// TIA Portal project "XC221_TRABALHO_FINAL" (V13)

(* hardware
DEVICE "S7-1200 station_1"  SIMATIC 1200-Station
   slot 0: "S7-1200 rack"  Rack  V1.0
   slot 1: "PLC_123"  CPU 1214C DC/DC/DC  6ES7 214-1AG31-0XB0  V3.0
   slot 3: "AQ1 x 12 bits"  6ES7 232-4HA30-0XB0  V1.0
*)

// ===== PLC "PLC_123"  CPU 1214C DC/DC/DC =====
// protected blocks, not shown: "EASYPI", "MEMRST"

VAR_GLOBAL   // PLC tag table "Default tag table"
   "System_Byte" AT %MB1 : Byte;
   "FirstScan" AT %M1.0 : Bool;   // Primeiro Scan do sistema
   "DiagStatusUpdate" AT %M1.1 : Bool;
   "AlwaysTRUE" AT %M1.2 : Bool;   // Usado para manter o sistema ligado sempre
   "AlwaysFALSE" AT %M1.3 : Bool;   // Usado para manter o sistema desligado sempre
   "Clock_Byte" AT %MB0 : Byte;
   "Clock_10Hz" AT %M0.0 : Bool;
   "Clock_5Hz" AT %M0.1 : Bool;
   "Clock_2.5Hz" AT %M0.2 : Bool;
   "Clock_2Hz" AT %M0.3 : Bool;
   "Clock_1.25Hz" AT %M0.4 : Bool;
   "Clock_1Hz" AT %M0.5 : Bool;
   "Clock_0.625Hz" AT %M0.6 : Bool;
   "Clock_0.5Hz" AT %M0.7 : Bool;
END_VAR

VAR_GLOBAL   // PLC tag table "01- Entradas Digitais"
   "DIn_GERAL_Emerge" AT %I0.0 : Bool;   // Ativa condição de emergência
   "DIn_GERAL_Rearma" AT %I0.1 : Bool;   // Rearma defeitos
   "DIn_GERAL_SelLoc" AT %I0.2 : Bool;   // Seleciona local (válvula e ventiladores)
   "DIn_VS101_Abre" AT %I0.3 : Bool;   // Botão abre válvula
   "DIn_VS101_Fecha" AT %I0.4 : Bool;   // Botão fecha válvula
   "DIn_VT101_LigDsg" AT %I0.5 : Bool;   // Botao liga/desliga ventilador 1
   "DIn_VT102_LigDsg" AT %I0.6 : Bool;   // Botao liga/desliga ventilador 2
   "DIn_BA101_DisjOff" AT %I0.7 : Bool;   // Disjuntor da bomba desarmado
END_VAR

VAR_GLOBAL   // PLC tag table "02- Saidas Digitais"
   "DOu_VS101_Abre" AT %Q0.0 : Bool;   // Abre válvula (energiza)
   "DOu_VT101_Liga" AT %Q0.1 : Bool;   // Liga ventilador 1 (energiza)
   "DOu_VT102_Liga" AT %Q0.2 : Bool;   // Liga ventilador 2 (energiza)
END_VAR

VAR_GLOBAL   // PLC tag table "03-Entradas Analogicas"
   "AIn_LT101_Nivel" AT %IW64 : UInt;   // Nível de água no tanque [bruto]
END_VAR

VAR_GLOBAL   // PLC tag table "04-Saidas Analogicas"
   "AOu_BA101_VelBmb" AT %QW64 : UInt;   // Velocidade da bomba [bruto]
END_VAR

VAR_GLOBAL   // PLC tag table "05-Comandos"
   "Cmd_GERAL_Rearma" AT %M101.0 : Bool;   // Rearma defeitos
   "Cmd_VS101_Abre" AT %M102.0 : Bool;   // Abre válvula
   "Cmd_VS101_Fecha" AT %M102.1 : Bool;   // Fecha válvula
   "Cmd_VT101_Liga" AT %M103.0 : Bool;   // Liga ventilador 1
   "Cmd_VT101_Deslig" AT %M103.1 : Bool;   // Desliga ventilador 1
   "Cmd_VT101_HorRst" AT %M103.2 : Bool;   // Zera horímetro do ventilador 1
   "Cmd_VT102_Liga" AT %M104.0 : Bool;   // Liga ventilador 2
   "Cmd_VT102_Deslig" AT %M104.1 : Bool;   // Desliga ventilador 2
   "Cmd_VT102_HorRst" AT %M104.2 : Bool;   // Zera horímetro do ventilador 2
   "Cmd_BA101_Liga" AT %M108.0 : Bool;   // Liga bomba
   "Cmd_BA101_Deslig" AT %M108.1 : Bool;   // Desliga bomba
   "Cmd_BA101_HorRst" AT %M108.2 : Bool;   // Zera horímetro da bomba
   "Cmd_BA101_SelMan" AT %M108.3 : Bool;   // Seleciona modo “Manual” da bomba
   "Cmd_BA101_SelAut" AT %M108.4 : Bool;   // Seleciona modo “Automático” da bomba
   "Cmd_BA101_SelPID" AT %M108.5 : Bool;   // Seleciona modo “PID” da bomba
   "Cmd BA101 SelOnOff" AT %M108.6 : Bool;   // Seleciona modo “On/Off” da bomba
END_VAR

VAR_GLOBAL   // PLC tag table "06-Estados"
   "Stt_GERAL_LocSel" AT %M201.0 : Bool;   // Local selecionado (válvula e ventiladores)
   "Stt_VS101_Aberta" AT %M202.0 : Bool;   // Válvula aberta (energizada)
   "Stt_VT101_Ligado" AT %M203.0 : Bool;   // Ventilador 1 ligado
   "Stt_VT101_Defeito" AT %M203.1 : Bool;   // Ventilador 1 com defeito
   "Stt_VT102_Ligado" AT %M204.0 : Bool;   // Ventilador 2 ligado
   "Stt_VT102_Defeito" AT %M204.1 : Bool;   // Ventilador 2 com defeito
   "Stt_LC101_LigBmb" AT %M206.0 : Bool;   // Solicitação do controlador On/Off para ligar bomba
   "Stt_BA101_Ligada" AT %M208.0 : Bool;   // Bomba ligada
   "Stt_BA101_Defeito" AT %M208.1 : Bool;   // Bomba com defeito
   "Stt_BA101_Bloq" AT %M208.2 : Bool;   // Bomba bloqueada
   "Stt_BA101_ManSel" AT %M208.3 : Bool;   // Bomba em modo “Manual”
   "Stt_BA101_PIDSel" AT %M208.4 : Bool;   // Bomba em modo “PID”
END_VAR

VAR_GLOBAL   // PLC tag table "07-Alarmes"
   "Alr_GERAL_Emerge" AT %M301.0 : Bool;   // Condição de emergência ativada
   "Alr_VT101_HorFim" AT %M303.0 : Bool;   // Ventilador 1 com horas esgotadas
   "Alr_VT102_HorFim" AT %M304.0 : Bool;   // Ventilador 2 com horas esgotadas
   "Alr_LT101_ExcedHH" AT %M305.0 : Bool;   // Limite “Muito Alto” excedido
   "Alr_LT101_ExcedH" AT %M305.1 : Bool;   // Limite “Alto” excedido
   "Alr_LT101_ExcedL" AT %M305.2 : Bool;   // Limite “Baixo” excedido
   "Alr_LT101_ExcedLL" AT %M305.3 : Bool;   // Limite “Muito Baixo” excedido
   "Alr_BA101_HorFim" AT %M308.0 : Bool;   // Bomba com horas esgotadas
   "Alr_BA101_DisjOff" AT %M308.1 : Bool;   // Disjuntor da bomba desarmado
END_VAR

VAR_GLOBAL   // PLC tag table "08-Auxiliares Digitais"
   "DAu_GERAL_Rearma" AT %M401.0 : Bool;   // Algum botão de rearme atuado
   "DAu_GERAL_Pul1s0" AT %M401.1 : Bool;   // Pulso de 1 scan a cada 1.0 segundo
   "DAu_VS101_AbrLoc" AT %M402.0 : Bool;   // Abre via modo local
   "DAu_VS101_AbrRem" AT %M402.1 : Bool;   // Abre via modo remoto
   "DAu_VT101_LigLoc" AT %M403.0 : Bool;   // Liga via modo local
   "DAu_VT101_LigRem" AT %M403.1 : Bool;   // Liga via modo remoto
   "DAu_VT101_EdgLig" AT %M403.2 : Bool;   // Borda para ligar ventilador 1
   "DAu_VT101_EdgDsg" AT %M403.3 : Bool;   // Borda para desligar ventilador 1
   "DAu_VT102_LigLoc" AT %M404.0 : Bool;   // Liga via modo local
   "DAu_VT102_LigRem" AT %M404.1 : Bool;   // Liga via modo remoto
   "DAu_VT102_EdgLig" AT %M404.2 : Bool;   // Borda para ligar ventilador 2
   "DAu_VT102_EdgDsg" AT %M404.3 : Bool;   // Borda para desligar ventilador 2
   "DAu_BA101_LigMan" AT %M408.0 : Bool;   // Liga via modo manual
   "DAu_BA101_LigOnOff" AT %M408.1 : Bool;   // Liga via modo On/Off
   "DAu_BA101_LigPID" AT %M408.2 : Bool;   // Liga via modo PID
END_VAR

VAR_GLOBAL   // PLC tag table "09-Auxiliares Analógicos"
   "AAu_VT101_Horas" AT %MD505 : Real;   // Horas trabalhadas do ventilador 1
   "AAu_VT101_Minutos" AT %MD509 : Real;   // Minutos trabalhados do ventilador 1
   "AAu_VT101_Segs" AT %MD513 : Real;   // Segundos trabalhados do ventilador 1
   "AAu_VT102_Horas" AT %MD517 : Real;   // Horas trabalhadas do ventilador 2
   "AAu_VT102_Minutos" AT %MD521 : Real;   // Minutos trabalhados do ventilador 2
   "AAu_VT102_Segs" AT %MD525 : Real;   // Segundos trabalhados do ventilador 2
   "AAu_LT101_NivelFP" AT %MD533 : Real;   // Nıvel em formato real [bruto]
   "AAu_LC102_LstErr" AT %MD553 : Real;   // Último valor de erro
   "AAu_LC102_LstInt" AT %MD557 : Real;   // Último valor da ação integral
   "AAu_BA101_Horas" AT %MD537 : Real;   // Horas trabalhadas da bomba
   "AAu_BA101_Minutos" AT %MD541 : Real;   // Minutos trabalhados da bomba
   "AAu_BA101_Segs" AT %MD545 : Real;   // Segundos trabalhados da bomba
   "AAu_BA101_VelBmb" AT %MD549 : Real;   // Velocidade em formato real [bruto]
END_VAR

VAR_GLOBAL   // PLC tag table "10-Analógicas"
   "Ana_GERAL_AtvCPU" AT %MD601 : Real;   // Sinalizador de atividade da CPU
   "Ana_VT101_HorDec" AT %MD605 : Real;   // Horas restantes do ventilador 1
   "Ana_VT102_HorDec" AT %MD619 : Real;   // Horas restantes do ventilador 2
   "Ana_LT101_Nivel" AT %MD613 : Real;   // Nível de água no tanque [mm]
   "Ana_LC102_SinCtrl" AT %MD617 : Real;   // Sinal de controle [%]
   "Ana_BA101_HorDec" AT %MD621 : Real;   // Horas restantes da bomba
   "Ana_BA101_VelBmb" AT %MD625 : Real;   // Velocidade atual da bomba [%]
END_VAR

VAR_GLOBAL   // PLC tag table "11-Parâmetros"
   "Par_VT101_HorLim" AT %MD705 : Real;   // Limite de horas do ventilador 1
   "Par_VT102_HorLim" AT %MD709 : Real;   // Limite de horas do ventilador 2
   "Par_LT101_LimHH" AT %MD713 : Real;   // Limite para a condição “Muito Alto” [mm]
   "Par_LT101_LimH" AT %MD717 : Real;   // Limite para a condição “Alto” [mm]
   "Par_LT101_LimL" AT %MD721 : Real;   // Limite para a condição “Baixo” [mm]
   "Par_LT101_LimLL" AT %MD725 : Real;   // Limite para a condição “Muito Baixo” [mm]
   "Par_LC101_LimDsg" AT %MD729 : Real;   // Limite para desligar a bomba [mm]
   "Par_LC101_LimLig" AT %MD733 : Real;   // Limite para ligar a bomba [mm]
   "Par_LC102_Setpoint" AT %MD737 : Real;   // Setpoint [mm]
   "Par_LC102_Prop" AT %MD741 : Real;   // Ganho proporcional
   "Par_LC102_Integ" AT %MD745 : Real;   // Tempo integral [segundos]
   "Par_BA101_HorLim" AT %MD753 : Real;   // Limite de horas da bomba
   "Par_BA101_RefVel" AT %MD757 : Real;   // Referência de velocidade da bomba [%]
END_VAR

DATA_BLOCK "AUXPRG"   // DB1
TITLE = Variáveis auxiliares para programação
{ S7_Optimized_Access := 'FALSE' }
AUTHOR : Dimitri
VERSION : 0.1
// Posições de memória para uso em temporizadores, contadores, instruções de detecção de borda etc.
   VAR
      "Timer" : Array [1 .. 20] of IEC_TIMER;
      "Counter" : Array [1 .. 20] of IEC_COUNTER;
      Edge : Array [1 .. 20] of Bool;
   END_VAR
BEGIN
END_DATA_BLOCK

DATA_BLOCK "HORIM_DB"   // DB6
{ S7_Optimized_Access := 'FALSE' }
VERSION : 0.1
// stored: InstanceOfName HORIM
"HORIM"
BEGIN
END_DATA_BLOCK

DATA_BLOCK "Vetor_Array"   // DB7
{ S7_Optimized_Access := 'FALSE' }
VERSION : 0.1
   VAR
      Borda : Array[0..3] of Bool;
   END_VAR
BEGIN
END_DATA_BLOCK

// folder: System blocks/Program resources

DATA_BLOCK "IEC_Timer_0_DB"   // DB2
{ S7_Optimized_Access := 'FALSE' }
AUTHOR : Simatic
FAMILY : IEC
NAME : IEC_TMR
VERSION : 1.0
// stored: InstanceOfName ?
"?"
BEGIN
END_DATA_BLOCK

DATA_BLOCK "IEC_Counter_0_DB"   // DB3
{ S7_Optimized_Access := 'FALSE' }
AUTHOR : Simatic
FAMILY : IEC
NAME : CNTR
VERSION : 1.0
// stored: InstanceOfName ?
"?"
BEGIN
END_DATA_BLOCK

DATA_BLOCK "IEC_Timer_0_DB_0"   // DB4
{ S7_Optimized_Access := 'FALSE' }
AUTHOR : Simatic
FAMILY : IEC
NAME : IEC_TMR
VERSION : 1.0
// stored: InstanceOfName ?
"?"
BEGIN
END_DATA_BLOCK

DATA_BLOCK "IEC_Counter_0_DB_1"   // DB5
{ S7_Optimized_Access := 'FALSE' }
AUTHOR : Simatic
FAMILY : IEC
NAME : CNTR
VERSION : 1.0
// stored: InstanceOfName ?
"?"
BEGIN
END_DATA_BLOCK

// folder: (top level)

FUNCTION_BLOCK "HORIM"   // FB1, LAD
TITLE = Horímetro
{ S7_Optimized_Access := 'FALSE' }
VERSION : 0.1
   VAR_TEMP   // added for the SCL form of the ladder/FBD networks
      _w1 : Bool;
   END_VAR
BEGIN

REGION Network 1: Segundos
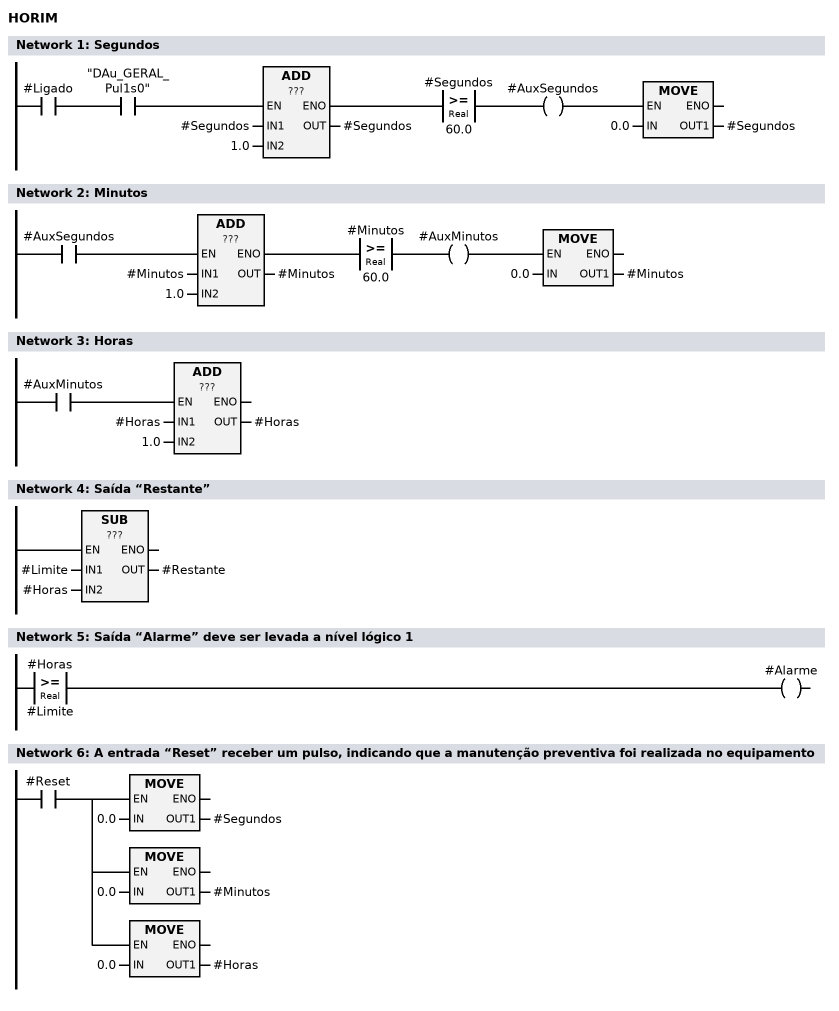
   RUNG wire#powerrail
      Contact( #Ligado )
      Contact( "DAu_GERAL_Pul1s0" )
      { S7_Templates := "SrcType := ???"; S7_GenerateENO := "TRUE" } Add(in1 := #Segundos, in2 := 1.0, out => #Segundos)
      { S7_Templates := "SrcType := Real" } GE_Contact(in1 := #Segundos, in2 := 60.0)
      Coil( #AuxSegundos )
      { S7_GenerateENO := "TRUE" } Move(in := 0.0, out1 => #Segundos)
   END_RUNG
   // the same network as SCL:
   // ENO of a box is taken as its EN; it also drops when the box reports an error
   #_w1 := #Ligado AND "DAu_GERAL_Pul1s0";
   IF #_w1 THEN #Segundos := #Segundos + 1.0; END_IF;
   #AuxSegundos := #_w1 AND (#Segundos >= 60.0);
   IF #AuxSegundos THEN #Segundos := 0.0; END_IF;
END_REGION

REGION Network 2: Minutos
   RUNG wire#powerrail
      Contact( #AuxSegundos )
      { S7_Templates := "SrcType := ???"; S7_GenerateENO := "TRUE" } Add(in1 := #Minutos, in2 := 1.0, out => #Minutos)
      { S7_Templates := "SrcType := Real" } GE_Contact(in1 := #Minutos, in2 := 60.0)
      Coil( #AuxMinutos )
      { S7_GenerateENO := "TRUE" } Move(in := 0.0, out1 => #Minutos)
   END_RUNG
   // the same network as SCL:
   // ENO of a box is taken as its EN; it also drops when the box reports an error
   IF #AuxSegundos THEN #Minutos := #Minutos + 1.0; END_IF;
   #AuxMinutos := #AuxSegundos AND (#Minutos >= 60.0);
   IF #AuxMinutos THEN #Minutos := 0.0; END_IF;
END_REGION

REGION Network 3: Horas
   RUNG wire#powerrail
      Contact( #AuxMinutos )
      { S7_Templates := "SrcType := ???"; S7_GenerateENO := "TRUE" } Add(in1 := #Horas, in2 := 1.0, out => #Horas)
   END_RUNG
   // the same network as SCL:
   IF #AuxMinutos THEN #Horas := #Horas + 1.0; END_IF;
END_REGION

REGION Network 4: Saída “Restante”
   RUNG wire#powerrail
      { S7_Templates := "SrcType := ???"; S7_GenerateENO := "TRUE" } Sub(in1 := #Limite, in2 := #Horas, out => #Restante)
   END_RUNG
   // the same network as SCL:
   #Restante := #Limite - #Horas;
END_REGION

REGION Network 5: Saída “Alarme” deve ser levada a nível lógico 1
   RUNG wire#powerrail
      { S7_Templates := "SrcType := Real" } GE_Contact(in1 := #Horas, in2 := #Limite)
      Coil( #Alarme )
   END_RUNG
   // the same network as SCL:
   #Alarme := #Horas >= #Limite;
END_REGION

REGION Network 6: A entrada “Reset” receber um pulso, indicando que a manutenção preventiva foi realizada no equipamento
   RUNG wire#powerrail
      Contact( #Reset )
      wire#w1
      { S7_GenerateENO := "TRUE" } Move(in := 0.0, out1 => #Segundos)
   END_RUNG
   RUNG wire#w1
      { S7_GenerateENO := "TRUE" } Move(in := 0.0, out1 => #Minutos)
   END_RUNG
   RUNG wire#w1
      { S7_GenerateENO := "TRUE" } Move(in := 0.0, out1 => #Horas)
   END_RUNG
   // the same network as SCL:
   IF #Reset THEN
       #Segundos := 0.0;
       #Minutos := 0.0;
       #Horas := 0.0;
   END_IF;
END_REGION
END_FUNCTION_BLOCK

FUNCTION "GERAL" : Void   // FC1, LAD
TITLE = Elemento 1 (Elementos Gerais do Sistema)
{ S7_Optimized_Access := 'FALSE' }
VERSION : 0.1
// Descrição funcional: o grupo em questão abrange todos os elementos do sistema. Seu propósito é gerar sinais (estados, alarmes etc) considerados comuns a esses elementos. A implementação desses sinais deverá respeitar as especificações a seguir.
BEGIN

REGION Network 1: Condição de emergência ativada (Alarme)
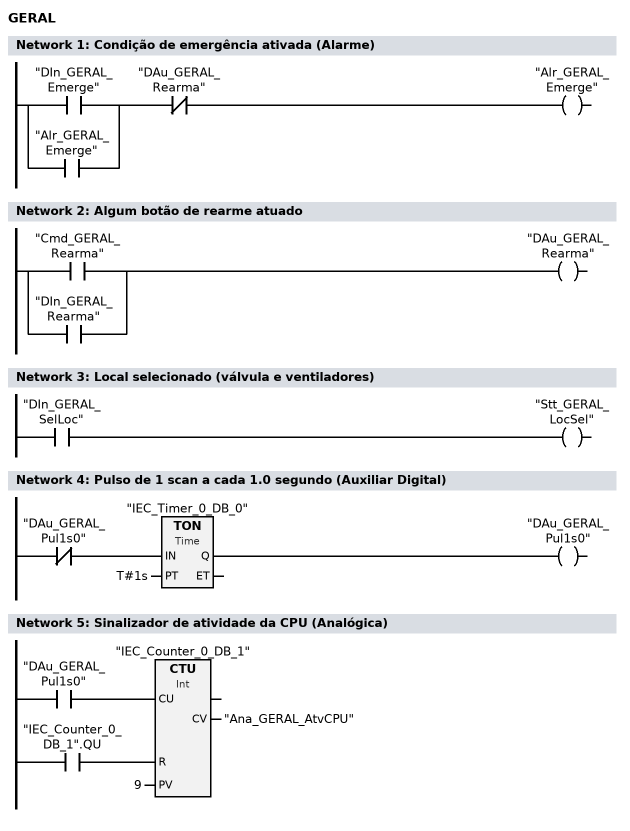
   RUNG wire#powerrail
      Contact( "DIn_GERAL_Emerge" )
      wire#w1
      I_Contact( "DAu_GERAL_Rearma" )
      Coil( "Alr_GERAL_Emerge" )
   END_RUNG
   RUNG wire#powerrail
      Contact( "Alr_GERAL_Emerge" )
   END_RUNG wire#w1
   // the same network as SCL:
   "Alr_GERAL_Emerge" := ("DIn_GERAL_Emerge" OR "Alr_GERAL_Emerge") AND NOT "DAu_GERAL_Rearma";
END_REGION

REGION Network 2: Algum botão de rearme atuado
   RUNG wire#powerrail
      Contact( "Cmd_GERAL_Rearma" )
      wire#w1
      Coil( "DAu_GERAL_Rearma" )
   END_RUNG
   RUNG wire#powerrail
      Contact( "DIn_GERAL_Rearma" )
   END_RUNG wire#w1
   // the same network as SCL:
   "DAu_GERAL_Rearma" := "Cmd_GERAL_Rearma" OR "DIn_GERAL_Rearma";
END_REGION

REGION Network 3: Local selecionado (válvula e ventiladores)
   RUNG wire#powerrail
      Contact( "DIn_GERAL_SelLoc" )
      Coil( "Stt_GERAL_LocSel" )
   END_RUNG
   // the same network as SCL:
   "Stt_GERAL_LocSel" := "DIn_GERAL_SelLoc";
END_REGION

REGION Network 4: Pulso de 1 scan a cada 1.0 segundo (Auxiliar Digital)
   "IEC_Timer_0_DB_0".TON(IN := NOT "DAu_GERAL_Pul1s0", PT := T#1s);
   "DAu_GERAL_Pul1s0" := "IEC_Timer_0_DB_0".Q;
END_REGION

REGION Network 5: Sinalizador de atividade da CPU (Analógica)
   "IEC_Counter_0_DB_1".CTU(CU := "DAu_GERAL_Pul1s0",
                           R := "IEC_Counter_0_DB_1".QU,
                           PV := 9,
                           CV => "Ana_GERAL_AtvCPU");
END_REGION
END_FUNCTION

FUNCTION "VS101" : Void   // FC2, LAD
TITLE = Elemento 2 (Válvula Solenóide)
{ S7_Optimized_Access := 'FALSE' }
VERSION : 0.1
// Descrição funcional: este equipamento tem a função de controlar o fluxo de água entre os reservatórios superior e inferior. Sua operação pode ocorrer por meio de dois modos excludentes: local ou remoto. Na verdade, essa seleção é realizada no grupo “Elementos Gerais do Sistema”. Isto é, a válvula deverá assumir o modo de operação indicado por uma variável do referido grupo.
BEGIN

REGION Network 1: Abre via modo local (Auxiliar Digital)
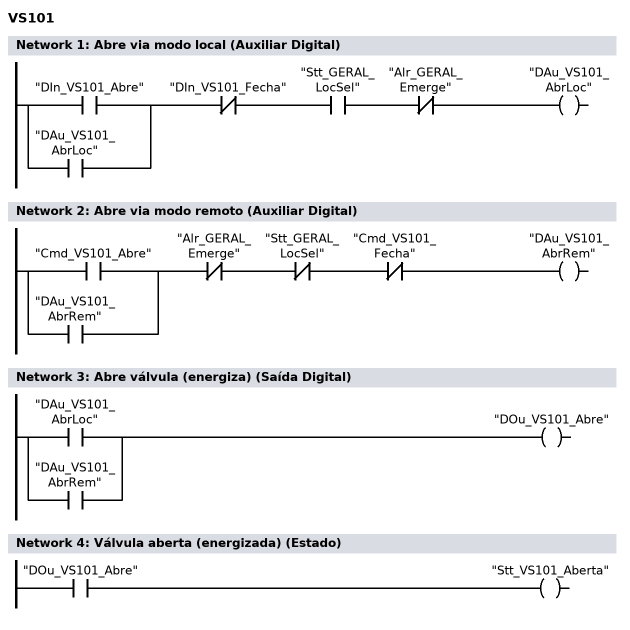
   RUNG wire#powerrail
      Contact( "DIn_VS101_Abre" )
      wire#w1
      I_Contact( "DIn_VS101_Fecha" )
      Contact( "Stt_GERAL_LocSel" )
      I_Contact( "Alr_GERAL_Emerge" )
      Coil( "DAu_VS101_AbrLoc" )
   END_RUNG
   RUNG wire#powerrail
      Contact( "DAu_VS101_AbrLoc" )
   END_RUNG wire#w1
   // the same network as SCL:
   "DAu_VS101_AbrLoc" := ("DIn_VS101_Abre" OR "DAu_VS101_AbrLoc") AND NOT "DIn_VS101_Fecha" AND "Stt_GERAL_LocSel" AND NOT "Alr_GERAL_Emerge";
END_REGION

REGION Network 2: Abre via modo remoto (Auxiliar Digital)
   RUNG wire#powerrail
      Contact( "Cmd_VS101_Abre" )
      wire#w1
      I_Contact( "Alr_GERAL_Emerge" )
      I_Contact( "Stt_GERAL_LocSel" )
      I_Contact( "Cmd_VS101_Fecha" )
      Coil( "DAu_VS101_AbrRem" )
   END_RUNG
   RUNG wire#powerrail
      Contact( "DAu_VS101_AbrRem" )
   END_RUNG wire#w1
   // the same network as SCL:
   "DAu_VS101_AbrRem" := ("Cmd_VS101_Abre" OR "DAu_VS101_AbrRem") AND NOT "Alr_GERAL_Emerge" AND NOT "Stt_GERAL_LocSel" AND NOT "Cmd_VS101_Fecha";
END_REGION

REGION Network 3: Abre válvula (energiza) (Saída Digital)
   RUNG wire#powerrail
      Contact( "DAu_VS101_AbrLoc" )
      wire#w1
      Coil( "DOu_VS101_Abre" )
   END_RUNG
   RUNG wire#powerrail
      Contact( "DAu_VS101_AbrRem" )
   END_RUNG wire#w1
   // the same network as SCL:
   "DOu_VS101_Abre" := "DAu_VS101_AbrLoc" OR "DAu_VS101_AbrRem";
END_REGION

REGION Network 4: Válvula aberta (energizada) (Estado)
   RUNG wire#powerrail
      Contact( "DOu_VS101_Abre" )
      Coil( "Stt_VS101_Aberta" )
   END_RUNG
   // the same network as SCL:
   "Stt_VS101_Aberta" := "DOu_VS101_Abre";
END_REGION
END_FUNCTION

FUNCTION "VT101" : Void   // FC3, LAD
TITLE = Elemento 3 (Ventilador 1)
{ S7_Optimized_Access := 'FALSE' }
VERSION : 0.1
// Descrição funcional: este equipamento não está instalado fisicamente na planta, mas tem a função de permitir a implementação de alguns conceitos importantes de programação. A entrada digital associada a ele está conectada a um botão comum, similarmente aos demais equipamentos da planta. Porém, a saída digital que deveria acionar um motor, está conectada a um LED, que simulará seu funcionamento. Sua operação pode ocorrer por meio de dois modos excludentes: local ou remoto. Na verdade, essa seleção é realizada no grupo “Elementos Gerais do Sistema”. Isto é, o ventilador deverá assumir o modo de operação indicado por uma varíavel do referido grupo.
   VAR_TEMP   // added for the SCL form of the ladder/FBD networks
      _w1 : Bool;
   END_VAR
BEGIN

REGION Network 1: Horas restantes do ventilador 1 (Analógica) e Ventilador 1 com horas esgotadas (Alarme)
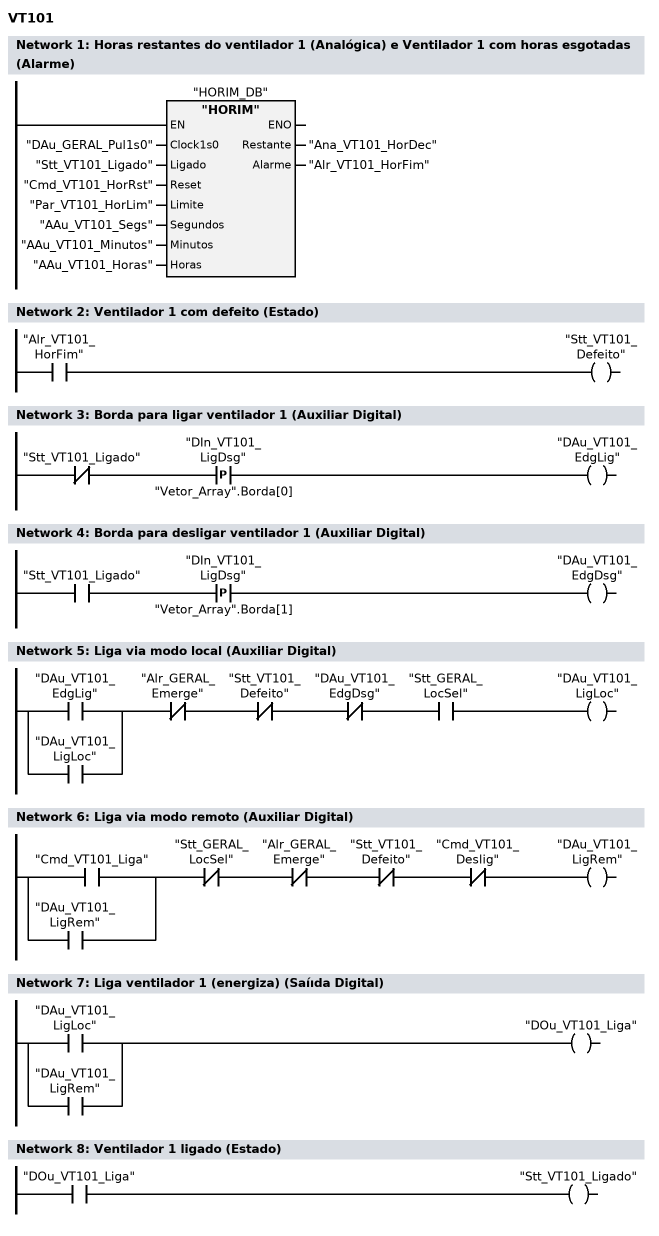
   RUNG wire#powerrail
      "HORIM_DB"(Clock1s0 := "DAu_GERAL_Pul1s0", Ligado := "Stt_VT101_Ligado", Reset := "Cmd_VT101_HorRst", Limite := "Par_VT101_HorLim", Segundos := "AAu_VT101_Segs", Minutos := "AAu_VT101_Minutos", Horas := "AAu_VT101_Horas", Restante => "Ana_VT101_HorDec", Alarme => "Alr_VT101_HorFim")
   END_RUNG
   // the same network as SCL:
   "HORIM_DB"(Clock1s0 := "DAu_GERAL_Pul1s0",   // "HORIM"
              Ligado := "Stt_VT101_Ligado",
              Reset := "Cmd_VT101_HorRst",
              Limite := "Par_VT101_HorLim",
              Segundos := "AAu_VT101_Segs",
              Minutos := "AAu_VT101_Minutos",
              Horas := "AAu_VT101_Horas",
              Restante => "Ana_VT101_HorDec",
              Alarme => "Alr_VT101_HorFim");
END_REGION

REGION Network 2: Ventilador 1 com defeito (Estado)
   RUNG wire#powerrail
      Contact( "Alr_VT101_HorFim" )
      Coil( "Stt_VT101_Defeito" )
   END_RUNG
   // the same network as SCL:
   "Stt_VT101_Defeito" := "Alr_VT101_HorFim";
END_REGION

REGION Network 3: Borda para ligar ventilador 1 (Auxiliar Digital)
   RUNG wire#powerrail
      I_Contact( "Stt_VT101_Ligado" )
      P_Contact(operand := "DIn_VT101_LigDsg", bit := "Vetor_Array".Borda[0])
      Coil( "DAu_VT101_EdgLig" )
   END_RUNG
   // the same network as SCL:
   #_w1 := NOT "Stt_VT101_Ligado" AND "DIn_VT101_LigDsg" AND NOT "Vetor_Array".Borda[0];   // rising edge of "DIn_VT101_LigDsg"
   "Vetor_Array".Borda[0] := "DIn_VT101_LigDsg";
   "DAu_VT101_EdgLig" := #_w1;
END_REGION

REGION Network 4: Borda para desligar ventilador 1 (Auxiliar Digital)
   RUNG wire#powerrail
      Contact( "Stt_VT101_Ligado" )
      P_Contact(operand := "DIn_VT101_LigDsg", bit := "Vetor_Array".Borda[1])
      Coil( "DAu_VT101_EdgDsg" )
   END_RUNG
   // the same network as SCL:
   #_w1 := "Stt_VT101_Ligado" AND "DIn_VT101_LigDsg" AND NOT "Vetor_Array".Borda[1];   // rising edge of "DIn_VT101_LigDsg"
   "Vetor_Array".Borda[1] := "DIn_VT101_LigDsg";
   "DAu_VT101_EdgDsg" := #_w1;
END_REGION

REGION Network 5: Liga via modo local (Auxiliar Digital)
   RUNG wire#powerrail
      Contact( "DAu_VT101_EdgLig" )
      wire#w1
      I_Contact( "Alr_GERAL_Emerge" )
      I_Contact( "Stt_VT101_Defeito" )
      I_Contact( "DAu_VT101_EdgDsg" )
      Contact( "Stt_GERAL_LocSel" )
      Coil( "DAu_VT101_LigLoc" )
   END_RUNG
   RUNG wire#powerrail
      Contact( "DAu_VT101_LigLoc" )
   END_RUNG wire#w1
   // the same network as SCL:
   "DAu_VT101_LigLoc" := ("DAu_VT101_EdgLig" OR "DAu_VT101_LigLoc") AND NOT "Alr_GERAL_Emerge" AND NOT "Stt_VT101_Defeito" AND NOT "DAu_VT101_EdgDsg" AND "Stt_GERAL_LocSel";
END_REGION

REGION Network 6: Liga via modo remoto (Auxiliar Digital)
   RUNG wire#powerrail
      Contact( "Cmd_VT101_Liga" )
      wire#w1
      I_Contact( "Stt_GERAL_LocSel" )
      I_Contact( "Alr_GERAL_Emerge" )
      I_Contact( "Stt_VT101_Defeito" )
      I_Contact( "Cmd_VT101_Deslig" )
      Coil( "DAu_VT101_LigRem" )
   END_RUNG
   RUNG wire#powerrail
      Contact( "DAu_VT101_LigRem" )
   END_RUNG wire#w1
   // the same network as SCL:
   "DAu_VT101_LigRem" := ("Cmd_VT101_Liga" OR "DAu_VT101_LigRem") AND NOT "Stt_GERAL_LocSel" AND NOT "Alr_GERAL_Emerge" AND NOT "Stt_VT101_Defeito" AND NOT "Cmd_VT101_Deslig";
END_REGION

REGION Network 7: Liga ventilador 1 (energiza) (Saíıda Digital)
   RUNG wire#powerrail
      Contact( "DAu_VT101_LigLoc" )
      wire#w1
      Coil( "DOu_VT101_Liga" )
   END_RUNG
   RUNG wire#powerrail
      Contact( "DAu_VT101_LigRem" )
   END_RUNG wire#w1
   // the same network as SCL:
   "DOu_VT101_Liga" := "DAu_VT101_LigLoc" OR "DAu_VT101_LigRem";
END_REGION

REGION Network 8: Ventilador 1 ligado (Estado)
   RUNG wire#powerrail
      Contact( "DOu_VT101_Liga" )
      Coil( "Stt_VT101_Ligado" )
   END_RUNG
   // the same network as SCL:
   "Stt_VT101_Ligado" := "DOu_VT101_Liga";
END_REGION
END_FUNCTION

FUNCTION "VT102" : Void   // FC3, LAD
TITLE = Elemento 4 (Ventilador 2)
{ S7_Optimized_Access := 'FALSE' }
VERSION : 0.1
// Descrição funcional: este equipamento não está instalado fisicamente na planta, mas tem a função de permitir a implementação de alguns conceitos importantes de programação. A entrada digital associada a ele está conectada a um botão comum, similarmente aos demais equipamentos da planta. Porém, a saída digital que deveria acionar um motor, está conectada a um LED, que simulará seu funcionamento. Sua operação pode ocorrer por meio de dois modos excludentes: local ou remoto. Na verdade, essa seleção é realizada no grupo “Elementos Gerais do Sistema”. Isto é, o ventilador deverá assumir o modo de operação indicado por uma varíavel do referido grupo.
   VAR_TEMP   // added for the SCL form of the ladder/FBD networks
      _w1 : Bool;
   END_VAR
BEGIN

REGION Network 1: Horas restantes do ventilador 1 (Analógica) e Ventilador 1 com horas esgotadas (Alarme)
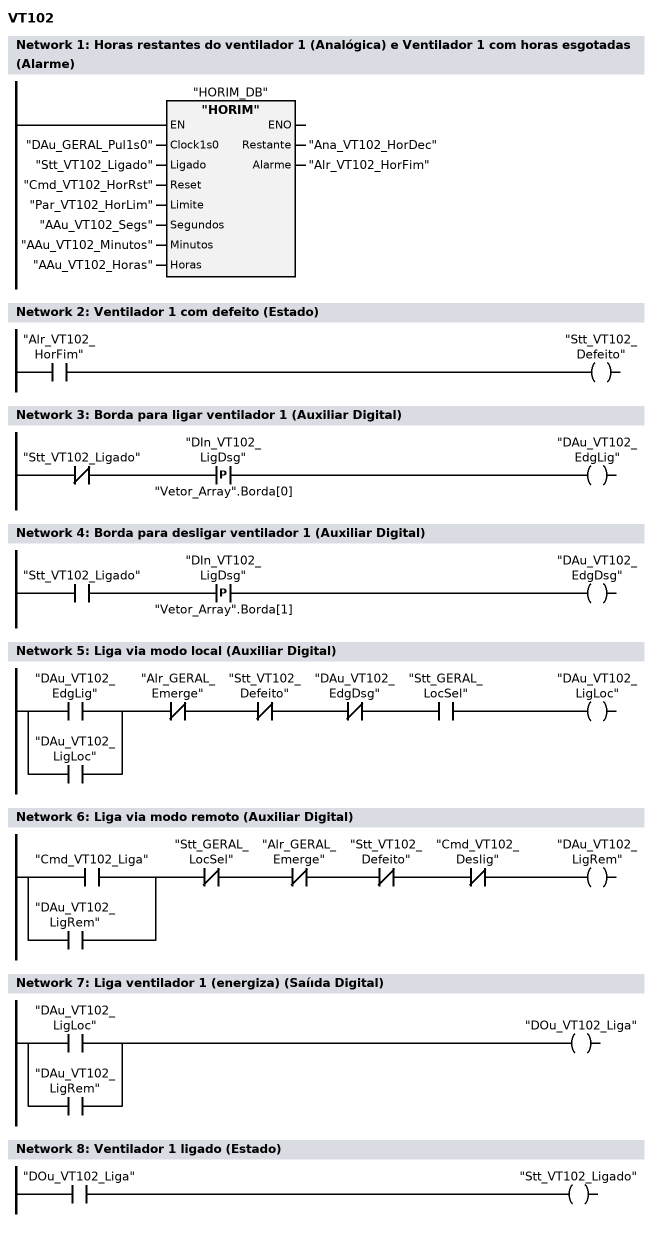
   RUNG wire#powerrail
      "HORIM_DB"(Clock1s0 := "DAu_GERAL_Pul1s0", Ligado := "Stt_VT102_Ligado", Reset := "Cmd_VT102_HorRst", Limite := "Par_VT102_HorLim", Segundos := "AAu_VT102_Segs", Minutos := "AAu_VT102_Minutos", Horas := "AAu_VT102_Horas", Restante => "Ana_VT102_HorDec", Alarme => "Alr_VT102_HorFim")
   END_RUNG
   // the same network as SCL:
   "HORIM_DB"(Clock1s0 := "DAu_GERAL_Pul1s0",   // "HORIM"
              Ligado := "Stt_VT102_Ligado",
              Reset := "Cmd_VT102_HorRst",
              Limite := "Par_VT102_HorLim",
              Segundos := "AAu_VT102_Segs",
              Minutos := "AAu_VT102_Minutos",
              Horas := "AAu_VT102_Horas",
              Restante => "Ana_VT102_HorDec",
              Alarme => "Alr_VT102_HorFim");
END_REGION

REGION Network 2: Ventilador 1 com defeito (Estado)
   RUNG wire#powerrail
      Contact( "Alr_VT102_HorFim" )
      Coil( "Stt_VT102_Defeito" )
   END_RUNG
   // the same network as SCL:
   "Stt_VT102_Defeito" := "Alr_VT102_HorFim";
END_REGION

REGION Network 3: Borda para ligar ventilador 1 (Auxiliar Digital)
   RUNG wire#powerrail
      I_Contact( "Stt_VT102_Ligado" )
      P_Contact(operand := "DIn_VT102_LigDsg", bit := "Vetor_Array".Borda[0])
      Coil( "DAu_VT102_EdgLig" )
   END_RUNG
   // the same network as SCL:
   #_w1 := NOT "Stt_VT102_Ligado" AND "DIn_VT102_LigDsg" AND NOT "Vetor_Array".Borda[0];   // rising edge of "DIn_VT102_LigDsg"
   "Vetor_Array".Borda[0] := "DIn_VT102_LigDsg";
   "DAu_VT102_EdgLig" := #_w1;
END_REGION

REGION Network 4: Borda para desligar ventilador 1 (Auxiliar Digital)
   RUNG wire#powerrail
      Contact( "Stt_VT102_Ligado" )
      P_Contact(operand := "DIn_VT102_LigDsg", bit := "Vetor_Array".Borda[1])
      Coil( "DAu_VT102_EdgDsg" )
   END_RUNG
   // the same network as SCL:
   #_w1 := "Stt_VT102_Ligado" AND "DIn_VT102_LigDsg" AND NOT "Vetor_Array".Borda[1];   // rising edge of "DIn_VT102_LigDsg"
   "Vetor_Array".Borda[1] := "DIn_VT102_LigDsg";
   "DAu_VT102_EdgDsg" := #_w1;
END_REGION

REGION Network 5: Liga via modo local (Auxiliar Digital)
   RUNG wire#powerrail
      Contact( "DAu_VT102_EdgLig" )
      wire#w1
      I_Contact( "Alr_GERAL_Emerge" )
      I_Contact( "Stt_VT102_Defeito" )
      I_Contact( "DAu_VT102_EdgDsg" )
      Contact( "Stt_GERAL_LocSel" )
      Coil( "DAu_VT102_LigLoc" )
   END_RUNG
   RUNG wire#powerrail
      Contact( "DAu_VT102_LigLoc" )
   END_RUNG wire#w1
   // the same network as SCL:
   "DAu_VT102_LigLoc" := ("DAu_VT102_EdgLig" OR "DAu_VT102_LigLoc") AND NOT "Alr_GERAL_Emerge" AND NOT "Stt_VT102_Defeito" AND NOT "DAu_VT102_EdgDsg" AND "Stt_GERAL_LocSel";
END_REGION

REGION Network 6: Liga via modo remoto (Auxiliar Digital)
   RUNG wire#powerrail
      Contact( "Cmd_VT102_Liga" )
      wire#w1
      I_Contact( "Stt_GERAL_LocSel" )
      I_Contact( "Alr_GERAL_Emerge" )
      I_Contact( "Stt_VT102_Defeito" )
      I_Contact( "Cmd_VT102_Deslig" )
      Coil( "DAu_VT102_LigRem" )
   END_RUNG
   RUNG wire#powerrail
      Contact( "DAu_VT102_LigRem" )
   END_RUNG wire#w1
   // the same network as SCL:
   "DAu_VT102_LigRem" := ("Cmd_VT102_Liga" OR "DAu_VT102_LigRem") AND NOT "Stt_GERAL_LocSel" AND NOT "Alr_GERAL_Emerge" AND NOT "Stt_VT102_Defeito" AND NOT "Cmd_VT102_Deslig";
END_REGION

REGION Network 7: Liga ventilador 1 (energiza) (Saíıda Digital)
   RUNG wire#powerrail
      Contact( "DAu_VT102_LigLoc" )
      wire#w1
      Coil( "DOu_VT102_Liga" )
   END_RUNG
   RUNG wire#powerrail
      Contact( "DAu_VT102_LigRem" )
   END_RUNG wire#w1
   // the same network as SCL:
   "DOu_VT102_Liga" := "DAu_VT102_LigLoc" OR "DAu_VT102_LigRem";
END_REGION

REGION Network 8: Ventilador 1 ligado (Estado)
   RUNG wire#powerrail
      Contact( "DOu_VT102_Liga" )
      Coil( "Stt_VT102_Ligado" )
   END_RUNG
   // the same network as SCL:
   "Stt_VT102_Ligado" := "DOu_VT102_Liga";
END_REGION
END_FUNCTION

FUNCTION "LT101" : Void   // FC4, LAD
TITLE = Elemento 5 (Nível de Agua no Tanque)
{ S7_Optimized_Access := 'FALSE' }
VERSION : 0.1
// Descrição funcional: o instrumento em questão tem a função de medir o nível de água no reservatório superior. Caso os limites estipulados para essa grandeza sejam excedidos, os respectivos sinais de alarme devem ser gerados, possibilitando a apresentação de mensagens aos operadores por meio de sistemas externos.
BEGIN

REGION Network 1: Nível de água no tanque [mm] (Analógica)
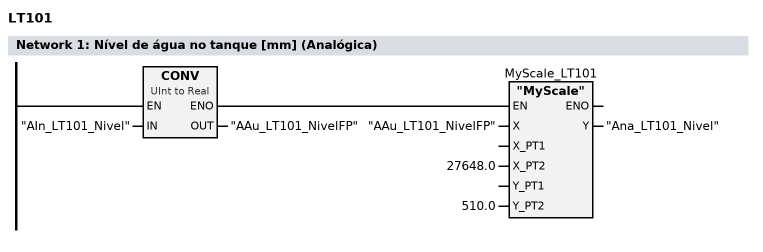
   RUNG wire#powerrail
      { S7_Templates := "[SrcType := UInt, DestType := Real]"; S7_GenerateENO := "TRUE" } Convert(in := "AIn_LT101_Nivel", out => "AAu_LT101_NivelFP")
      MyScale_LT101(X := "AAu_LT101_NivelFP", X_PT1 :=, X_PT2 := 27648.0, Y_PT1 :=, Y_PT2 := 510.0, Y => "Ana_LT101_Nivel")
   END_RUNG
   // the same network as SCL:
   // ENO of a box is taken as its EN; it also drops when the box reports an error
   "AAu_LT101_NivelFP" := UINT_TO_REAL("AIn_LT101_Nivel");
   MyScale_LT101(X := "AAu_LT101_NivelFP", X_PT2 := 27648.0, Y_PT2 := 510.0, Y => "Ana_LT101_Nivel");   // "MyScale"
END_REGION
END_FUNCTION

ORGANIZATION_BLOCK "Main"   // OB1, LAD, ProgramCycle
TITLE = Ciclo principal do programa
{ S7_Optimized_Access := 'FALSE' }
VERSION : 0.1
   VAR_TEMP   // added for the SCL form of the ladder/FBD networks
      _w1 : Bool;
      _w2 : Bool;
   END_VAR
BEGIN

REGION Network 1: Primeiro Scan do sistema
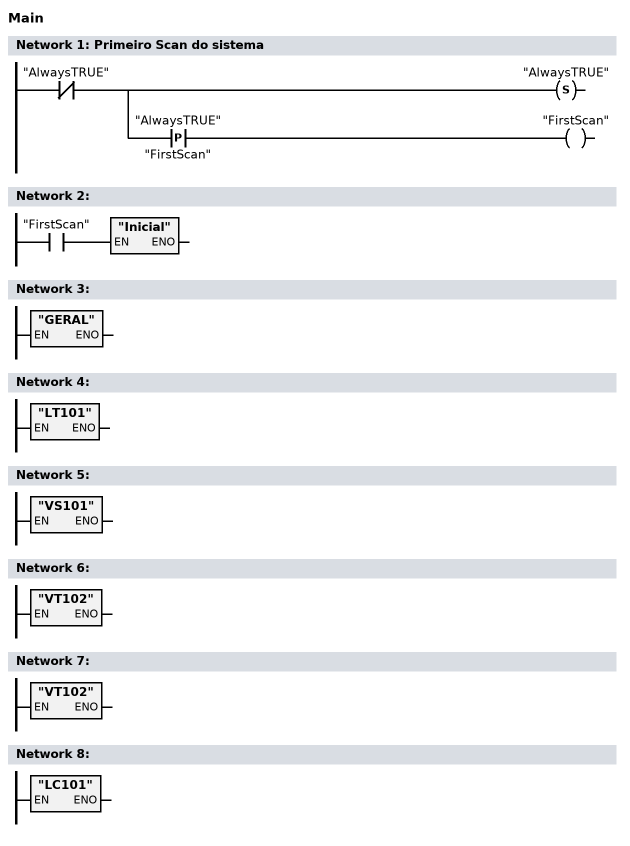
   RUNG wire#powerrail
      I_Contact( "AlwaysTRUE" )
      wire#w1
      S_Coil( "AlwaysTRUE" )
   END_RUNG
   RUNG wire#w1
      P_Contact(operand := "AlwaysTRUE", bit := "FirstScan")
      Coil( "FirstScan" )
   END_RUNG
   // the same network as SCL:
   #_w1 := NOT "AlwaysTRUE";
   IF #_w1 THEN "AlwaysTRUE" := TRUE; END_IF;
   #_w2 := #_w1 AND "AlwaysTRUE" AND NOT "FirstScan";   // rising edge of "AlwaysTRUE"
   "FirstScan" := "AlwaysTRUE";
   "FirstScan" := #_w2;
END_REGION

REGION Network 2
   RUNG wire#powerrail
      Contact( "FirstScan" )
      "Inicial"()
   END_RUNG
   // the same network as SCL:
   IF "FirstScan" THEN "Inicial"(); END_IF;
END_REGION

REGION Network 3
   RUNG wire#powerrail
      "GERAL"()
   END_RUNG
   // the same network as SCL:
   "GERAL"();
END_REGION

REGION Network 4
   RUNG wire#powerrail
      "LT101"()
   END_RUNG
   // the same network as SCL:
   "LT101"();
END_REGION

REGION Network 5
   RUNG wire#powerrail
      "VS101"()
   END_RUNG
   // the same network as SCL:
   "VS101"();
END_REGION

REGION Network 6
   RUNG wire#powerrail
      "VT102"()
   END_RUNG
   // the same network as SCL:
   "VT102"();
END_REGION

REGION Network 7
   RUNG wire#powerrail
      "VT102"()
   END_RUNG
   // the same network as SCL:
   "VT102"();
END_REGION

REGION Network 8
   RUNG wire#powerrail
      "LC101"()
   END_RUNG
   // the same network as SCL:
   "LC101"();
END_REGION
END_ORGANIZATION_BLOCK